Staubli VAL3: remSetnGlobal.pgx

program remSetnGlobal(string& sArgs[] (dimensions=1), num& nGlobal[] (dimensions=1), num nMin (dimensions=1), num nMax (dimensions=1), string sCmd (dimensions=1), string& sReturn[] (dimensions=1))
  local bool bOk
  local num nVal
begin
  // Read a command to set an arbitrary global value,
  // and respond accordingly.
  //
  logMsg("call remSetnGlobal")
  toNum(sArgs,nVal,bOk)
  if bOk
    if nVal<nMin
      nVal=nMin
    elseIf nVal>nMax
      nVal=nMax
    endIf
    nGlobal=nVal
    sReturn=sCmd+" "+toString(sNumConv,nGlobal)
  else
    call remErrNum(sCmd,sArgs,sReturn)
  endIf
end
